ABB RAPID module: 0034BD04

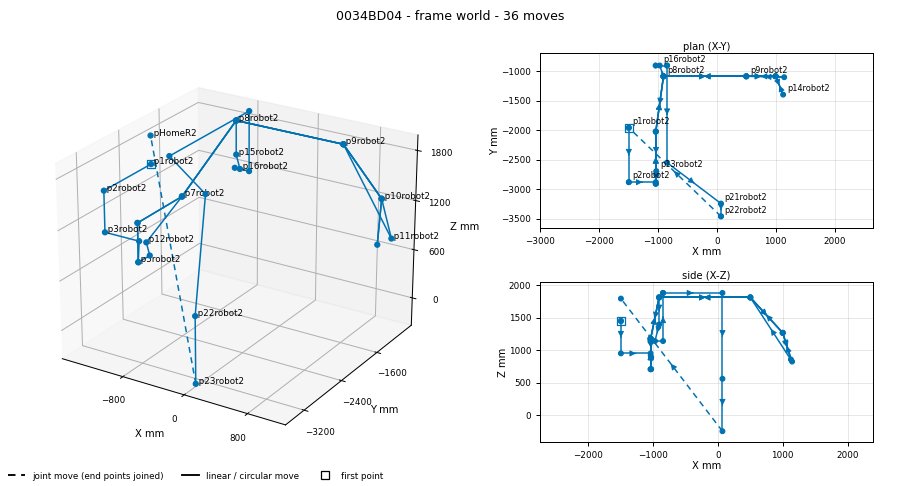
[picture p0: tool path of 0034BD04 in frame world, 36 of 36 moves have a stored position in this frame; points joined in program order, loops and branches not executed]
MODULE Module1
	CONST robtarget p1robot2:=[[-1492.73,-1959.33,1451.54],[1.38356E-30,-0.999996,-4.14231E-31,-0.00286655],[0,-1,0,0],[9E+09,9E+09,9E+09,9E+09,9E+09,9E+09]];
	CONST robtarget p2robot2:=[[-1492.73,-2882.81,1451.54],[4.88115E-09,0.999996,-1.01911E-09,0.00286655],[0,0,0,0],[9E+09,9E+09,9E+09,9E+09,9E+09,9E+09]];
	CONST robtarget p3robot2:=[[-1492.73,-2882.81,952.83],[0.00204012,0.702459,-0.711719,0.00201365],[0,0,1,0],[9E+09,9E+09,9E+09,9E+09,9E+09,9E+09]];
	CONST robtarget p4robot2:=[[-1035.11,-2882.81,952.83],[0.00204022,0.702458,-0.711719,0.00201364],[0,0,1,0],[9E+09,9E+09,9E+09,9E+09,9E+09,9E+09]];
	CONST robtarget p5robot2:=[[-1035.11,-2906.84,708.27],[0.00204025,0.702459,-0.711719,0.00201364],[0,0,1,0],[9E+09,9E+09,9E+09,9E+09,9E+09,9E+09]];
	CONST robtarget p6robot2:=[[-1035.11,-2906.84,1179.31],[0.00204017,0.702459,-0.711719,0.00201364],[0,0,1,0],[9E+09,9E+09,9E+09,9E+09,9E+09,9E+09]];
	CONST robtarget p7robot2:=[[-1035.11,-2023.99,1179.31],[0.304301,0.636728,-0.643388,-0.296697],[0,-1,1,0],[9E+09,9E+09,9E+09,9E+09,9E+09,9E+09]];
	CONST robtarget p8robot2:=[[-904.35,-1086.19,1814.83],[0.0235789,0.0663482,0.902757,0.424349],[-1,-1,1,0],[9E+09,9E+09,9E+09,9E+09,9E+09,9E+09]];
	CONST robtarget p9robot2:=[[500.46,-1086.19,1814.83],[0.0235788,0.0663484,0.902757,0.424349],[-2,0,0,0],[9E+09,9E+09,9E+09,9E+09,9E+09,9E+09]];
	CONST robtarget p10robot2:=[[999.37,-1086.19,1269.68],[0.320078,0.692241,0.583244,0.279603],[-2,-1,2,0],[9E+09,9E+09,9E+09,9E+09,9E+09,9E+09]];
	CONST robtarget p11robot2:=[[1143.87,-1101.28,827.11],[0.370648,0.622584,0.596582,0.345106],[-2,-2,2,0],[9E+09,9E+09,9E+09,9E+09,9E+09,9E+09]];
	CONST robtarget p12robot2:=[[-1026.51,-2757.33,893.00],[0.0078393,0.733279,-0.679634,-0.0183696],[0,-1,1,0],[9E+09,9E+09,9E+09,9E+09,9E+09,9E+09]];
	CONST robtarget p13robot2:=[[-1026.51,-2694.95,710.35],[0.0139111,0.708139,-0.705835,-0.0119233],[0,-1,1,0],[9E+09,9E+09,9E+09,9E+09,9E+09,9E+09]];
	CONST robtarget p14robot2:=[[1125.85,-1396.86,858.78],[0.320368,0.575146,0.629661,0.412431],[-2,-2,2,0],[9E+09,9E+09,9E+09,9E+09,9E+09,9E+09]];
	CONST robtarget p15robot2:=[[-904.35,-1086.19,1397.30],[0.554626,-0.0460075,-0.828152,-0.0666182],[-1,0,0,0],[9E+09,9E+09,9E+09,9E+09,9E+09,9E+09]];
	CONST robtarget p16robot2:=[[-968.37,-903.18,1142.54],[0.509646,0.00671145,-0.86015,-0.0189035],[-1,0,0,0],[9E+09,9E+09,9E+09,9E+09,9E+09,9E+09]];
	CONST robtarget p17robot2:=[[-1038.62,-903.18,1142.54],[0.509646,0.00671166,-0.86015,-0.0189034],[-1,0,0,0],[9E+09,9E+09,9E+09,9E+09,9E+09,9E+09]];
	CONST robtarget p18robot2:=[[-843.65,-903.18,1142.54],[0.509646,0.00671155,-0.86015,-0.0189035],[-1,0,0,0],[9E+09,9E+09,9E+09,9E+09,9E+09,9E+09]];
	CONST robtarget p19robot2:=[[-843.65,-903.18,1883.89],[0.509646,0.00671175,-0.86015,-0.0189036],[-1,0,1,0],[9E+09,9E+09,9E+09,9E+09,9E+09,9E+09]];
	CONST robtarget p20robot2:=[[-843.65,-2550.77,1883.89],[0.509646,0.00671201,-0.86015,-0.0189038],[0,-1,2,0],[9E+09,9E+09,9E+09,9E+09,9E+09,9E+09]];
	CONST robtarget p21robot2:=[[71.29,-3245.15,1883.89],[0.375231,0.610361,-0.606105,0.345395],[1,-1,2,0],[9E+09,9E+09,9E+09,9E+09,9E+09,9E+09]];
	CONST robtarget p22robot2:=[[71.29,-3462.79,561.87],[0.00383777,0.716466,-0.69734,-0.0194532],[1,-1,2,0],[9E+09,9E+09,9E+09,9E+09,9E+09,9E+09]];
	CONST robtarget p23robot2:=[[71.29,-3462.79,-245.81],[0.0139078,0.716341,-0.697545,-0.00964972],[1,-1,2,0],[9E+09,9E+09,9E+09,9E+09,9E+09,9E+09]];
	CONST robtarget pHomeR2:=[[-1492.73,-1959.33,1796.86],[0,-0.866025,0,0.5],[0,0,0,0],[9E+09,9E+09,9E+09,9E+09,9E+09,9E+09]];
    PROC main()
        !Add your code here
        MoveJ p1robot2, v1000, z50, tool0;
        MoveL p2robot2, v1000, z50, tool0;
        MoveL p3robot2, v1000, z50, tool0;
        MoveL p4robot2, v1000, z50, tool0;
        MoveL p5robot2, v1000, fine, tool0;
        WaitTime 1;
        SetDO vacuum, 1;
        MoveL p6robot2, v1000, z50, tool0;
        MoveL p7robot2, v1000, z50, tool0;
        MoveL p8robot2, v1000, z50, tool0;
        MoveL p9robot2, v1000, z50, tool0;
        MoveL p10robot2, v1000, z50, tool0;
        MoveL p11robot2, v1000, fine, tool0;
        SetDO robot2, 1;
        WaitUntil robot1=1;
        SetDO vacuum, 0;
        MoveL p9robot2, v1000, z50, tool0;
        MoveL p8robot2, v1000, z50, tool0;
        MoveL p7robot2, v1000, z50, tool0;
        MoveL p12robot2, v1000, z50, tool0;
        MoveL p13robot2, v1000, fine, tool0;
        SetDO vacuum, 1;
        MoveL p5robot2, v1000, z50, tool0;
        MoveL p6robot2, v1000, z50, tool0;
        MoveL p7robot2, v1000, z50, tool0;
        MoveL p8robot2, v1000, z50, tool0;
        MoveL p9robot2, v1000, z50, tool0;
        MoveL p10robot2, v1000, z50, tool0;
        MoveL p14robot2, v1000, fine, tool0;
        SetDO robot1, 0;
        SetDO robot2, 1;
        WaitUntil robot1=1;
        SetDO vacuum, 0;
        MoveL p10robot2, v1000, z20, tool0;
        MoveL p9robot2, v1000, z20, tool0;
        MoveL p8robot2, v1000, z20, tool0;
        MoveL p15robot2, v1000, z20, tool0;
        MoveL p16robot2, v1000, z20, tool0;
        MoveL p17robot2, v1000, fine, tool0;
        SetDO vacuum, 1;
        MoveL p18robot2, v1000, z20, tool0;
        MoveL p19robot2, v1000, z20, tool0;
        MoveL p20robot2, v1000, z20, tool0;
        MoveL p21robot2, v1000, z20, tool0;
        MoveL p22robot2, v1000, z20, tool0;
        MoveL p23robot2, v1000, fine, tool0;
        SetDO vacuum, 0;
        MoveJ pHomeR2, v1000, fine, tool0;
        SetDO robot1, 0;
        EXIT;
    ENDPROC
ENDMODULE
